(* CODESYS project IceFeedMotor.xml

Project tree, tasks and I/O mapping:
  function block IceFeedMotor [LD]
*)

// IceFeedMotor
FUNCTION_BLOCK IceFeedMotor
VAR_INPUT
	Run: 				BOOL;				//
	Override: 			BOOL;				//
	OverrideMotor: 		BOOL;				//
END_VAR
VAR_OUTPUT
	MotorOutput: 		BOOL;				//
END_VAR
VAR
END_VAR

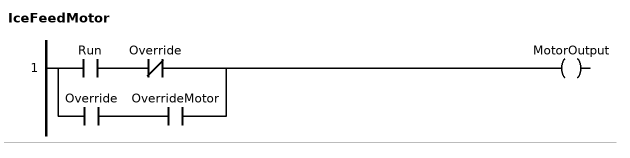
// NETWORK 1
MotorOutput := Run AND NOT Override OR Override AND OverrideMotor;

END_FUNCTION_BLOCK
